(* CoDeSys 2.3 export: STATION_7.EXP *)

(* POU STATION_7, FBD *)
FUNCTION_BLOCK STATION_7
VAR_INPUT
	xEMERGENCY								:	BOOL;
	xPB_START									:	BOOL;
	xSENSOR_ROTARY_STEP					:	BOOL;
	xSENSOR_PART_START_POS				:	BOOL;
	xSENSOR_PART_END_POS					:	BOOL;
	xSENSOR_PUNCH_PROXIMITY				:	BOOL;
	xSENSOR_PUNCH_FULLY_EXTENDED	:	BOOL;
	xSENSOR_DRILL_PROXIMITY				:	BOOL;
	xSENSOR_DRILL_UPPER_LIMIT			:	BOOL;
	xSENSOR_DRILL_LOWER_LIMIT			:	BOOL;
END_VAR
VAR_OUTPUT
	_xROTARY_MOTOR					:	BOOL;
	_xPUNCH								:	BOOL;
	_xLOWER_DRILL						:	BOOL;
	_xRAISE_DRILL						:	BOOL;
	_xDRILL								:	BOOL;
	_xDRILL_PUNCH						:	BOOL;
	_xIND_EMERGENCY					:	BOOL;
	_xIND_INIT_POS						:	BOOL;
	_xIND_PB_START					:	BOOL;
	_xIND_STATE_0						:	BOOL;
	_xIND_STATE_1						:	BOOL;
	_xIND_STATE_2						:	BOOL;
	_xIND_STATE_3						:	BOOL;
	_xIND_STATE_4						:	BOOL;
	_xIND_STATE_5						:	BOOL;
	_xIND_STATE_6						:	BOOL;
	_xIND_STATE_7						:	BOOL;
	_xIND_STATE_8						:	BOOL;
	_xFLAG_PROCESSING_PART		:	BOOL;
	_xFLAG_ACCEPT_NEW_PART		:	BOOL;
END_VAR
VAR
	calcTransitions			:	CALC_TRANSITIONS;
	seqCtrl					:	SEQUENTIAL_CTRL;
	actuatorCtrl				:	ACTUATOR_CTRL;
	calcFlags					:	CALC_FLAGS;
	indicatorCtrl				:	INDICATOR_CTRL;
END_VAR
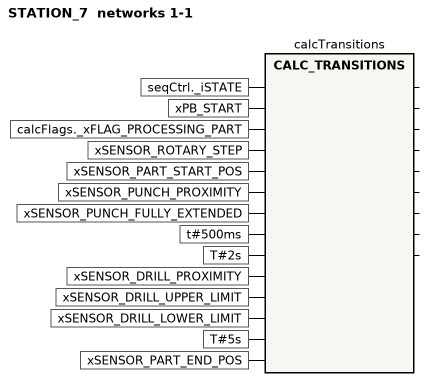
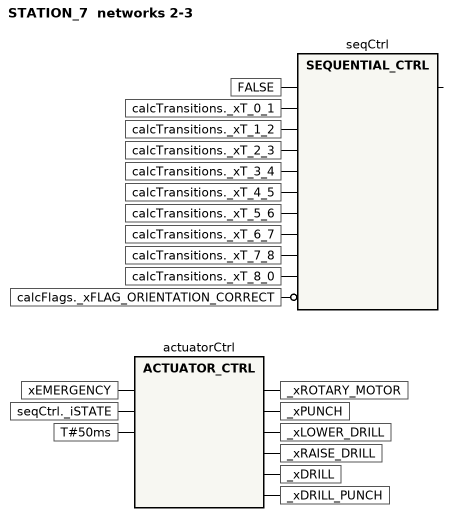
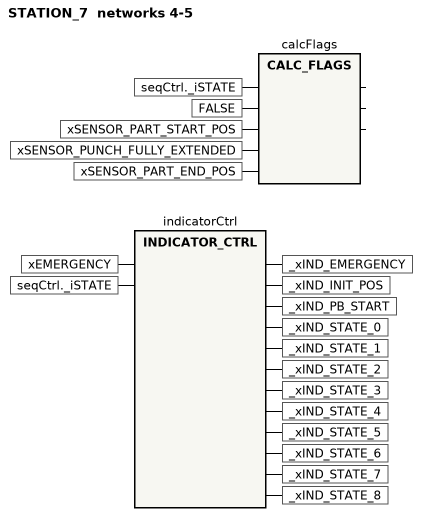
_FBD_ (* Function Block Diagram *)
NETWORK 1 transitions: (* Gets sensor values and calculates transitional conditions. *)
	calcTransitions:CALC_TRANSITIONS(seqCtrl._iSTATE, xPB_START, calcFlags._xFLAG_PROCESSING_PART, xSENSOR_ROTARY_STEP, xSENSOR_PART_START_POS, xSENSOR_PUNCH_PROXIMITY, xSENSOR_PUNCH_FULLY_EXTENDED, t#500ms, T#2s, xSENSOR_DRILL_PROXIMITY, xSENSOR_DRILL_UPPER_LIMIT, xSENSOR_DRILL_LOWER_LIMIT, T#5s, xSENSOR_PART_END_POS)
NETWORK 2 stateMachine: (* Saves and outputs the current machine state, increments if the corresponding transitional condition is met, returning back to state 0 from state 8. If the jump flag is set, steps 5,6 and 7 are skipped. *)
	seqCtrl:SEQUENTIAL_CTRL(FALSE, calcTransitions._xT_0_1, calcTransitions._xT_1_2, calcTransitions._xT_2_3, calcTransitions._xT_3_4, calcTransitions._xT_4_5, calcTransitions._xT_5_6, calcTransitions._xT_6_7, calcTransitions._xT_7_8, calcTransitions._xT_8_0, NOT calcFlags._xFLAG_ORIENTATION_CORRECT)
NETWORK 3 actuators: (* Controls which actuators are active in each state, all actuators get turned off in case of an emergency. *)
	actuatorCtrl:ACTUATOR_CTRL(xEMERGENCY, seqCtrl._iSTATE, T#50ms, out 2 => _xPUNCH, out 3 => _xLOWER_DRILL, out 4 => _xRAISE_DRILL, out 5 => _xDRILL, out 6 => _xDRILL_PUNCH) => _xROTARY_MOTOR
NETWORK 4 flags: (* Sets various flags for communication with other stations and between POUs of this station. *)
	calcFlags:CALC_FLAGS(seqCtrl._iSTATE, FALSE, xSENSOR_PART_START_POS, xSENSOR_PUNCH_FULLY_EXTENDED, xSENSOR_PART_END_POS)
NETWORK 5 stateIndicator: (* Lights corresponding light for each state (used mainly for debugging) *)
	indicatorCtrl:INDICATOR_CTRL(xEMERGENCY, seqCtrl._iSTATE, out 2 => _xIND_INIT_POS, out 3 => _xIND_PB_START, out 4 => _xIND_STATE_0, out 5 => _xIND_STATE_1, out 6 => _xIND_STATE_2, out 7 => _xIND_STATE_3, out 8 => _xIND_STATE_4, out 9 => _xIND_STATE_5, out 10 => _xIND_STATE_6, out 11 => _xIND_STATE_7, out 12 => _xIND_STATE_8) => _xIND_EMERGENCY
_END_FBD_
(* the same logic as Structured Text *)
(* Network 1 *)
calcTransitions(seqCtrl._iSTATE, xPB_START, calcFlags._xFLAG_PROCESSING_PART, xSENSOR_ROTARY_STEP, xSENSOR_PART_START_POS, xSENSOR_PUNCH_PROXIMITY, xSENSOR_PUNCH_FULLY_EXTENDED, t#500ms, T#2s, xSENSOR_DRILL_PROXIMITY, xSENSOR_DRILL_UPPER_LIMIT, xSENSOR_DRILL_LOWER_LIMIT, T#5s, xSENSOR_PART_END_POS);
(* Network 2 *)
seqCtrl(FALSE, calcTransitions._xT_0_1, calcTransitions._xT_1_2, calcTransitions._xT_2_3, calcTransitions._xT_3_4, calcTransitions._xT_4_5, calcTransitions._xT_5_6, calcTransitions._xT_6_7, calcTransitions._xT_7_8, calcTransitions._xT_8_0, NOT calcFlags._xFLAG_ORIENTATION_CORRECT);
(* Network 3: see the listing above *)
(* Network 4 *)
calcFlags(seqCtrl._iSTATE, FALSE, xSENSOR_PART_START_POS, xSENSOR_PUNCH_FULLY_EXTENDED, xSENSOR_PART_END_POS);
(* Network 5: see the listing above *)
END_FUNCTION_BLOCK
